// Struckig
// Copyright (C) 2022 Stefan Besler

// This program is free software: you can redistribute it and/or modify
// it under the terms of the GNU General Public License as published by
// the Free Software Foundation, either version 3 of the License, or
// (at your option) any later version.

// This program is distributed in the hope that it will be useful,
// but WITHOUT ANY WARRANTY; without even the implied warranty of
// MERCHANTABILITY or FITNESS FOR A PARTICULAR PURPOSE.  See the
// GNU General Public License for more details.
//
// You should have received a copy of the GNU General Public License
// along with THIS PROGRAM.  IF NOT, see <http://www.gnu.org/licenses/>.
{attribute 'conditionalshow'}
/// Positional envelope of a single-DoF profile.
/// The structure stores minimum/maximum position and the corresponding
/// times where these extrema occur along the generated trajectory.
///
/// It is returned by profile-bound checks to answer questions such as:
/// "What is the furthest negative/positive excursion and when does it happen?"
TYPE ProfileBound :
STRUCT
  Minimum, Maximum : LREAL; //< Extreme positions reached by the profile.
  Tmin, Tmax : LREAL;  //< Times at which `Minimum` and `Maximum` are reached.
END_STRUCT
END_TYPE

(* stored: Version 1.1.0.1
   DUT ProfileBound: Id {b615dcba-8544-436f-9a57-30985945064e} *)
